Fanuc KAREL source: kt00737.KL

-- PROVISIONAL review KL for V1013-1; original PC SHA256 fe4e4e0b5e3f9bf18eeb6e13c94985a73abafe89355cb2faa72c06e6dc0ae4d8
-- Incomplete behavior may be omitted. Consult companion uncertainty JSON. Do not deploy.
PROGRAM KT00737
%NOLOCKGROUP
BEGIN
  -- UNRESOLVED_PC offsets 5-18; opcodes 22,1D,23
  -- UNRESOLVED_PC offsets 23-27; opcodes 7F
END KT00737
